LIN {X 0,Y 29.617,Z 750.619,A -85,B 0,C 180,E1 -26499.908,E2 -26499.908} C_VEL
LIN {X 0,Y 33.916,Z 749.822,A -85,B 0,C 180,E1 -26508.985,E2 -26508.985} C_VEL
LIN {X 0,Y 22.242,Z 755.859,A -85,B 0,C 180,E1 -26528.893,E2 -26528.893} C_VEL
LIN {X 0,Y 16.487,Z 759.847,A -85,B 0,C 180,E1 -26567.611,E2 -26567.611} C_VEL
LIN {X 0,Y 20.242,Z 762.521,A -85,B 0,C 180,E1 -26612.691,E2 -26612.691} C_VEL
LIN {X 0,Y 32.997,Z 763.94,A -85,B 0,C 180,E1 -26638.369,E2 -26638.369} C_VEL
LIN {X 0,Y 47.514,Z 763.62,A -85,B 0,C 180,E1 -26648.585,E2 -26648.585} C_VEL
LIN {X 0,Y 31.019,Z 764.535,A -85,B 0,C 180,E1 -26660.867,E2 -26660.867} C_VEL
LIN {X 0,Y 18.891,Z 763.659,A -85,B 0,C 180,E1 -26690.614,E2 -26690.614} C_VEL
LIN {X 0,Y 16.629,Z 761.89,A -85,B 0,C 180,E1 -26730.037,E2 -26730.037} C_VEL
LIN {X 0,Y 20.9,Z 757.891,A -85,B 0,C 180,E1 -26775.9,E2 -26775.9} C_VEL
LIN {X 0,Y 24.287,Z 756.124,A -85,B 0,C 180,E1 -26785.468,E2 -26785.468} C_VEL
LIN {X 0,Y 22.456,Z 753.317,A -85,B 0,C 180,E1 -26822.561,E2 -26822.561} C_VEL
LIN {X 0,Y 22.534,Z 753.135,A -85,B 0,C 180,E1 -26826.427,E2 -26826.427} C_VEL
LIN {X 0,Y 22.022,Z 753.175,A -85,B 0,C 180,E1 -26833.317,E2 -26833.317} C_VEL
LIN {X 0,Y 20.063,Z 753.934,A -85,B 0,C 180,E1 -26842.079,E2 -26842.079} C_VEL
LIN {X 0,Y 16.567,Z 755.444,A -85,B 0,C 180,E1 -26853.811,E2 -26853.811} C_VEL
LIN {X 0,Y 12.133,Z 757.333,A -85,B 0,C 180,E1 -26870.671,E2 -26870.671} C_VEL
LIN {X 0,Y 7.838,Z 759.988,A -85,B 0,C 180,E1 -26923.724,E2 -26923.724} C_VEL
LIN {X 0,Y 11.235,Z 761.902,A -85,B 0,C 180,E1 -26977.82,E2 -26977.82} C_VEL
LIN {X 0,Y 25.265,Z 763.997,A -85,B 0,C 180,E1 -27008.54,E2 -27008.54} C_VEL
LIN {X 0,Y 10.805,Z 762.502,A -85,B 0,C 180,E1 -27042.332,E2 -27042.332} C_VEL
LIN {X 0,Y 8.617,Z 761.164,A -85,B 0,C 180,E1 -27090.072,E2 -27090.072} C_VEL
LIN {X 0,Y 15.028,Z 757.449,A -85,B 0,C 180,E1 -27153.86,E2 -27153.86} C_VEL
LIN {X 0,Y 15.112,Z 755.87,A -85,B 0,C 180,E1 -27190.148,E2 -27190.148} C_VEL
LIN {X 0,Y 20.854,Z 754.362,A -85,B 0,C 180,E1 -27224.692,E2 -27224.692} C_VEL
LIN {X 0,Y 9.615,Z 759.087,A -85,B 0,C 180,E1 -27263.966,E2 -27263.966} C_VEL
LIN {X 0,Y 11.235,Z 761.902,A -85,B 0,C 180,E1 -27337.82,E2 -27337.82} C_VEL
LIN {X 0,Y 10.709,Z 762.006,A -85,B 0,C 180,E1 -27344.283,E2 -27344.283} C_VEL
LIN {X 0,Y 8,Z 761.808,A -85,B 0,C 180,E1 -27352.722,E2 -27352.722} C_VEL
LIN {X 0,Y 3.029,Z 761.038,A -85,B 0,C 180,E1 -27366.726,E2 -27366.726} C_VEL
LIN {X 0,Y 0.837,Z 760.527,A -85,B 0,C 180,E1 -27357.359,E2 -27357.359} C_VEL
LIN {X 0,Y 7.884,Z 758.174,A -85,B 0,C 180,E1 -27203.675,E2 -27203.675} C_VEL
LIN {X 0,Y 6.733,Z 758.631,A -85,B 0,C 180,E1 -27182.877,E2 -27182.877} C_VEL
LIN {X 0,Y 1.096,Z 760.611,A -85,B 0,C 180,E1 -27025.581,E2 -27025.581} C_VEL
LIN {X 0,Y 1.485,Z 760.689,A -85,B 0,C 180,E1 -27009.801,E2 -27009.801} C_VEL
LIN {X 0,Y 0.837,Z 760.527,A -85,B 0,C 180,E1 -26997.359,E2 -26997.359} C_VEL
LIN {X 0,Y 1.794,Z 762.465,A -85,B 0,C 180,E1 -26856.976,E2 -26856.976} C_VEL
LIN {X 0,Y 1.794,Z 799,A -85,B 0,C 180,E1 -26856.976,E2 -26856.976} C_VEL
LIN {X 0,Y 1.794,Z 799,A -85,B 0,C 180,E1 -26856.976,E2 -26856.976}

QRS_NEXT_CUT()

QRS_NEXT()
QRS_HOME()

END
